RoboDK station: Assistive_UR5e.rdk

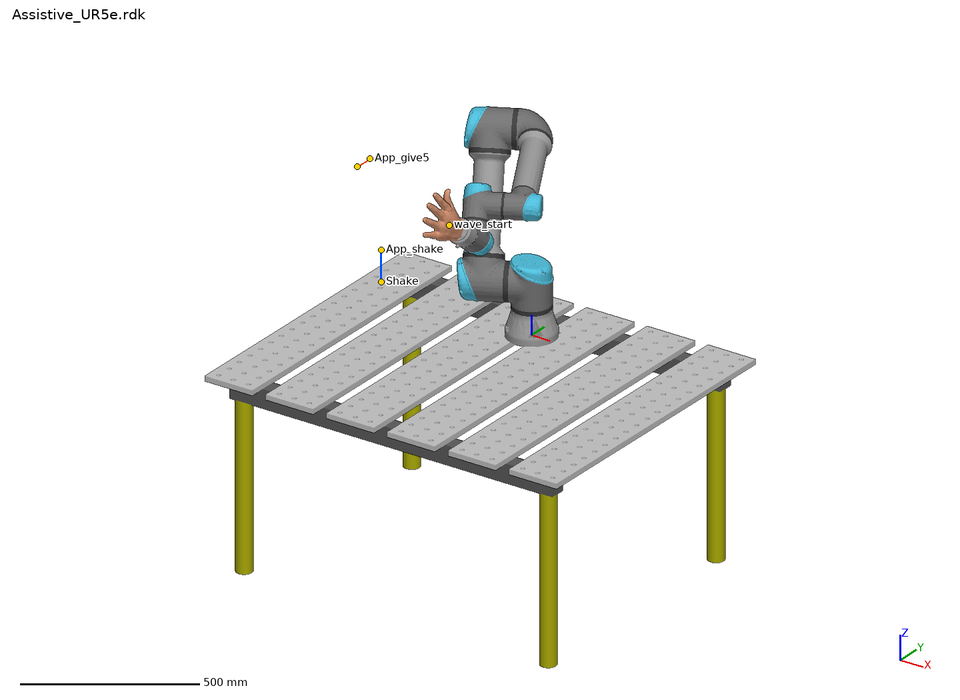
[picture v0: the station drawn from its stored meshes, robots at their saved joint values, targets as dots, program paths as lines]
Station Assistive_UR5e_SW (saved by RoboDK 5.9.2). Poses are relative to the parent item; angles as X-Y-Z fixed-axis rotations.
  - frame UR5e Base at (0, 0, 0) mm
    - robot UR5e: 6 axes, payload 5 kg, reach 850 mm, repeatability 0.03 mm, weight 18.4 kg
        modified DH rows (alpha deg, a mm, theta deg, d mm): 0, 0, 0, 162.5; 90, 0, 180, 0; 0, 425, 0, 0; 0, 392.25, 0, 133.3; -90, 0, 0, 99.7; 90, 0, 180, 99.6
        joint limits [-360, -360, -360, -360, -360, -360] to [360, 360, 360, 360, 360, 360]; home [0, -90, -90, 0, 90, 0]; saved at [-61.661, -60.826, -126.275, 227.863, -67.78, -18.055]
      - tool Hand, TCP at (0, 0, 50) mm, size 54.8 x 155.9 x 193.5 mm, geometry from Hand.stl
    - target wave_start (Cartesian target) at (0, -400, 500) mm, rotated rx 52.81 ry 0 rz 0 deg; joints [-61.661, -60.826, -126.275, 227.863, -67.78, -18.055] of UR5e
    - target wave_left (Cartesian target) at (0, -400, 500) mm, rotated rx -15.19 ry 0 rz 0 deg; joints [-72.332, -93.355, -127.409, 325.27, -94.562, -17.087] of UR5e
    - target wave_right (Cartesian target) at (0, -400, 500) mm, rotated rx 41.62 ry 0 rz 0 deg; joints [-63.68, -63.491, -130.157, 245.119, -72.874, -20.295] of UR5e
  - frame World at (0, 0, 0) mm
    - object Table at (0, 0, 0) mm, size 1193.8 x 965.2 x 609.6 mm, geometry from welding_table.sld
    - target Init (Cartesian target) at (0, -400, 500) mm, rotated rx 90 ry 0 rz 0 deg; joints [-57.836, -65.392, -107.167, 172.559, -57.836, 0] of UR5e
    - target App_shake (joint target) at (-300, -300, 300) mm, rotated rx 90 ry 0 rz 0 deg; joints [-129.97, -84.968, -123.366, -151.667, -129.97, 0] of UR5e
    - target Shake (joint target) at (-300, -300, 200) mm, rotated rx 90 ry 0 rz 0 deg; joints [-129.97, -95.332, -131.473, -133.195, -129.97, 0] of UR5e
    - target App_give5 (joint target) at (-380.86, -238.62, 533.82) mm, rotated rx 0 ry 0 rz 90 deg; joints [-130.679, -89.195, -122.013, 301.208, -90, 130.679] of UR5e
    - target Give5 (joint target) at (-380.86, -300, 533.82) mm, rotated rx 0 ry 0 rz 90 deg; joints [-125.814, -94.091, -116.939, 301.03, -90, 125.814] of UR5e
  - program Init (3 instructions, listed below)
  - program Hand_shake (5 instructions, listed below)
  - program Give_me_5! (5 instructions, listed below)
  - program MainProgram (4 instructions, listed below)
  - Python program sara Assistive_hand_SW_HW_sockets copy (listed below)
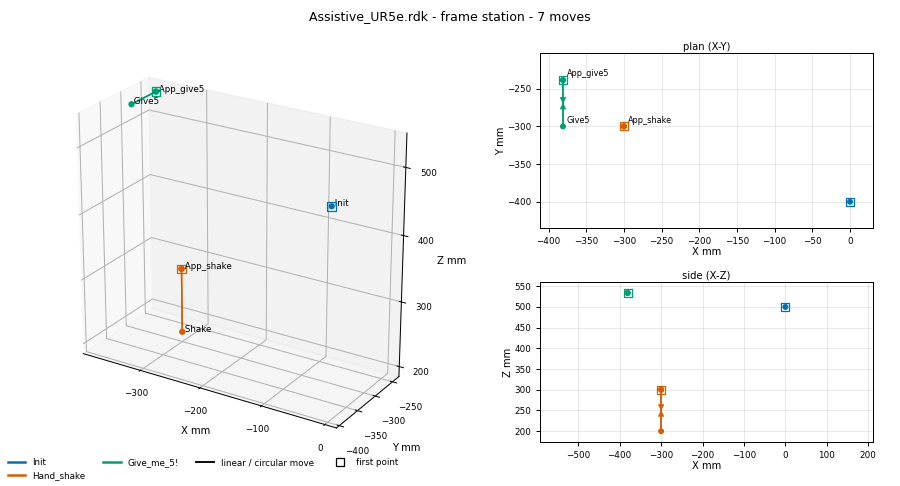
[picture p0: tool path of Assistive_UR5e.rdk in frame station, 7 of 7 moves have a stored position in this frame; points joined in program order, loops and branches not executed]

--- program Init (robot UR5e) ---
  Est. Ref.: UR5e Base
  Est. herr: Hand
  MoveJ (Init)

--- program Hand_shake (robot UR5e) ---
  Est. Ref.: UR5e Base
  Est. herr: Hand
  MoveL (App_shake)
  MoveL (Shake)
  MoveL (App_shake)

--- program Give_me_5! (robot UR5e) ---
  Est. Ref.: UR5e Base
  Est. herr: Hand
  MoveL (App_give5)
  MoveL (Give5)
  MoveL (App_give5)

--- program MainProgram (robot UR5e) ---
  Llamar Init
  Llamar Hand_shake
  Llamar Give_me_5!
  Llamar Init

--- Python program sara Assistive_hand_SW_HW_sockets copy ---
import os
import time
import socket
import tkinter as tk
from tkinter import messagebox
from math import radians, degrees, pi
import math
from robodk.robolink import *
from robodk.robomath import *

# Load RoboDK project from relative path
relative_path = "Assistive_UR5e.rdk"
absolute_path = os.path.abspath(relative_path)
RDK = Robolink()
# RDK.AddFile(absolute_path)

# Robot setup
robot = RDK.Item("UR5e")
base = RDK.Item("UR5e Base")
tool = RDK.Item('Hand')
Init_target = RDK.Item('Init')
wave_start_target = RDK.Item('wave_start')
wave_left_target = RDK.Item('wave_left')
wave_right_target = RDK.Item('wave_right')

robot.setPoseFrame(base)
robot.setPoseTool(tool)
robot.setSpeed(20)

# Robot Constants
ROBOT_IP = '192.168.1.5'
ROBOT_PORT = 30002
accel_mss = 1.2
speed_ms = 0.75
blend_r = 0.0
timej = 6
timel = 3

# URScript commands
set_tcp = "set_tcp(p[0.000000, 0.000000, 0.050000, 0.000000, 0.000000, 0.000000])"

deg_init = [-57.835746, -65.391528, -107.167117, 172.558645, -57.835746, 0.000000]
rad_init = [math.radians(j) for j in deg_init]
movej_init = f"movej({rad_init},{accel_mss},{speed_ms},{timel},0.0000)"

deg_start = [-61.661349, -60.826168, -126.275295, 227.862971, -67.780209, -18.054745]
rad_start =[math.radians(j) for j in deg_start]
movel_wave_start = f"movel({rad_start},{accel_mss},{speed_ms},{timel},0.000)"

deg_left = [-72.331751, -93.354688, -127.409127, 325.269567, -94.561656, -17.087400]
rad_left = [math.radians(j) for j in deg_left]
movel_wave_left = f"movel({rad_left},{accel_mss},{speed_ms},{timel/2},0.000)"

deg_right = [-63.680100, -63.491305, -130.156774, 245.118521, -72.874121, -20.294912]
rad_right = [math.radians(j) for j in deg_right]
movel_wave_right = f"movel({rad_right},{accel_mss},{speed_ms},{timel/2},0.000)"

# Check robot connection
def check_robot_port(ip, port):
    global robot_socket
    try:
        robot_socket = socket.socket(socket.AF_INET, socket.SOCK_STREAM)
        robot_socket.settimeout(1)
        robot_socket.connect((ip, port))
        return True
    except (socket.timeout, ConnectionRefusedError):
        return False
# Send URScript command
def send_ur_script(command):
    robot_socket.send((command + "\n").encode())


# Movements
def Init():
    print("Init")
    robot.MoveL(Init_target, True)
    print("Init_target REACHED")
    if robot_is_connected:
        print("Init REAL UR5e")
        send_ur_script(set_tcp)
        send_ur_script(movej_init)

def Wave():
    robot.MoveL(wave_start_target, True)
    for _ in range(3):
        robot.MoveL(wave_left_target, True)
        robot.MoveL(wave_right_target, True)
    robot.MoveL(wave_start_target, True)

    if robot_is_connected:
        send_ur_script(set_tcp)
        send_ur_script(movel_wave_left)
        send_ur_script(movel_wave_right)
        send_ur_script(movel_wave_left)


# Confirmation dialog to close RoboDK
def confirm_close():
    root = tk.Tk()
    root.withdraw()
    response = messagebox.askquestion(
        "Close RoboDK",
        "Do you want to save changes before closing RoboDK?",
        icon='question'
    )
    if response == 'yes':
        RDK.Save()
        RDK.CloseRoboDK()
        print("RoboDK saved and closed.")
    else:
        RDK.CloseRoboDK()
        print("RoboDK closed without saving.")

# Main function
def main():
    global robot_is_connected
    robot_is_connected = False
    Init()
    Wave()

# Run and close
if __name__ == "__main__":
    main()
    #confirm_close()
